
// ===== library: MasterCopy "APPLICATION_ID_READ_BLOCK" =====

FUNCTION_BLOCK "APPLICATION_ID_READ_BLOCK"   // FB5, SCL
{ S7_Optimized_Access := 'FALSE' }
VERSION : 0.1
   VAR_INPUT
      START_PARAMETER_READ : Bool;
      APPLICATION_ID : Int;
      PROFIdrive_OR_VACON_TELEGRAM_INPUT_ADDRESS : Int;
   END_VAR
   VAR_OUTPUT
      DONE : Bool;
      BUSY : Bool;
      ERROR : Bool;
      ERROR_CODE : DWord;
      VALUE : Int;
   END_VAR
   VAR
      PROFIdrive_param_read_request_record : Struct
         request_ref : Byte;
         request_id : Byte;
         axis_number : Byte;
         num_of_params_requested : Byte;
         attribute : Byte;
         num_of_elements : Byte;
         pnu : Int;
         subindex : Int;
      END_STRUCT;
      PROFIdrive_param_read_response : Struct
         request_ref : Byte;
         response_id : Byte;
         axis_number : Byte;
         num_of_parameters : Byte;
         format : Byte;
         num_of_values : Byte;
         value : Int;
      END_STRUCT;
      parameter_read_state : Int := 1;
      previous_start_parameter_read : Bool;
      stored_id : Int;
      stored_value : Int;
      WRREC_Instance : WRREC;
      stored_status : DWord;
      RDREC_Instance : RDREC;
      response_len : Int;
   END_VAR
   VAR_TEMP
      temp_done : Bool;
      temp_status : DWord;
      temp_error : Bool;
      temp_busy : Bool;
      temp_request_ref : Int;
      temp_valid : Bool;
      nooftries : Int;
   END_VAR
BEGIN
   CASE #parameter_read_state OF
       0:
           #parameter_read_state := 1;
           ;
       1:  // Statement section case 1
           IF #previous_start_parameter_read = 0 AND #START_PARAMETER_READ = 1 THEN
               #DONE := 0;
               #BUSY := 1;
               #ERROR := 0;
               #ERROR_CODE := 0;
               #nooftries := 0;
               #stored_id := #APPLICATION_ID;
               #PROFIdrive_param_read_request_record.attribute := 16#10;
               #PROFIdrive_param_read_request_record.axis_number := 1;
               #PROFIdrive_param_read_request_record.num_of_elements := 1;
               #PROFIdrive_param_read_request_record.num_of_params_requested := 1;
               #PROFIdrive_param_read_request_record.pnu := 10001;
               #PROFIdrive_param_read_request_record.request_id := 1; //change request, 1=read request
               #PROFIdrive_param_read_request_record.request_ref := INT_TO_CHAR(#temp_request_ref);
               #PROFIdrive_param_read_request_record.subindex := #stored_id;
               #temp_busy := 0;
               #temp_done := 0;
               #temp_error := 0;
               #temp_status := 0;
               #WRREC_Instance(REQ := 1,
                               ID := INT_TO_DWORD(#PROFIdrive_OR_VACON_TELEGRAM_INPUT_ADDRESS),
                               INDEX := 16#002f,
                               BUSY => #temp_busy,
                               DONE => #temp_done,
                               ERROR => #temp_error,
                               LEN := 10,
                               RECORD := #PROFIdrive_param_read_request_record,
                               STATUS => #stored_status);

               #parameter_read_state := 2; //start new parameter write sequence
           ELSE
               #parameter_read_state := 1;
               #DONE := 0;
               #BUSY := 0;
               #ERROR := 0;
               #ERROR_CODE := 0;
               #VALUE := 0;
           END_IF;
           ;
       2:  //check parameter write status
           #WRREC_Instance(REQ := 0,
                           ID := INT_TO_DWORD(#PROFIdrive_OR_VACON_TELEGRAM_INPUT_ADDRESS),
                           INDEX := 16#002f,
                           BUSY => #temp_busy,
                           DONE => #temp_done,
                           ERROR => #temp_error,
                           LEN := 10,
                           RECORD := #PROFIdrive_param_read_request_record,
                           STATUS => #stored_status);
           IF #temp_busy = 1 THEN
               // Statement section IF
               #parameter_read_state := 2; //check again next time
               #BUSY := 1;
               ;
           ELSIF #temp_done = 1 THEN
               #parameter_read_state := 3;
               #DONE := 0;
               #BUSY := 1;
               ;
           ELSIF #temp_error = 1 THEN
               #parameter_read_state := 20; //parameter write error state
               #ERROR := 1;
               #BUSY := 0;
               #ERROR_CODE := #stored_status;
           END_IF;
           ;

       3:  //Read response record
           #RDREC_Instance(REQ := 1,
                           ID := INT_TO_DWORD(#PROFIdrive_OR_VACON_TELEGRAM_INPUT_ADDRESS),
                           INDEX := 16#002f,
                           MLEN := 8,
                           BUSY => #temp_busy,
                           ERROR => #temp_error,
                           LEN => #response_len,
                           STATUS => #stored_status,
                           VALID => #temp_valid,
                           RECORD := #PROFIdrive_param_read_response);
           IF #temp_valid = 1 THEN
               // Statement section IF
               IF #PROFIdrive_param_read_response.format = 16#44 THEN
                   // Statement section IF
                   #parameter_read_state := 7; //done state
                   #DONE := 0;
                   #BUSY := 0;
                   #ERROR := 1;
                   #parameter_read_state := 30;
                   #VALUE := 0;
                   #ERROR_CODE := INT_TO_DWORD(#PROFIdrive_param_read_response.value);
                   #stored_status := #ERROR_CODE;
                   ;
               ELSE
                   #parameter_read_state := 7; //done state
                   #DONE := 1;
                   #BUSY := 0;
                   #VALUE := #PROFIdrive_param_read_response.value;
                   ;
               END_IF;
           ELSIF #temp_busy = 1 THEN
               #parameter_read_state := 3;
               #BUSY := 1;
               ;
           ELSIF #temp_error = 1 THEN
               IF #stored_status = 16#DE80B500 AND #nooftries < 10 THEN
                   #parameter_read_state := 4;
                   #DONE := 0;
                   #BUSY := 1;
                   #ERROR := 0;
                   #ERROR_CODE := 0;
                   #nooftries := #nooftries + 1;
                   ;
               ELSE
                   #parameter_read_state := 30;
                   #DONE := 0;
                   #BUSY := 0;
                   #ERROR := 1;
                   #ERROR_CODE := #stored_status;
                   ;
               END_IF;
               ;
           END_IF;
           ;
       4:
           //just a wait state when RDREC fails in state 3
           #parameter_read_state := 3;
           ;
       5:
           ;
       6:
           ;
       7:  // parameter write done state
           #DONE := 1;
           #BUSY := 0;
           #VALUE := #PROFIdrive_param_read_response.value;

           IF #START_PARAMETER_READ = 0 THEN
               // Statement section IF
               #parameter_read_state := 0;
               ;
           ELSE
               #parameter_read_state := 7;
           END_IF;

           ;
       20: //parameter write error state
           #BUSY := 0;
           #ERROR := 1;
           #DONE := 0;
           #ERROR_CODE := #stored_status;

           IF #START_PARAMETER_READ = 0 THEN
               // Statement section IF
               #parameter_read_state := 0;
               ;
           ELSE
               #parameter_read_state := 20;
           END_IF;

           ;
       30: //parameter write response error state
           #ERROR := 1;
           #ERROR_CODE := #stored_status;
           #DONE := 0;
           #BUSY := 0;

           IF #START_PARAMETER_READ = 0 THEN
               // Statement section IF
               #parameter_read_state := 0;
               ;
           ELSE
               #parameter_read_state := 30;
           END_IF;
           ;
       40:
           #BUSY := 0;
           #parameter_read_state := 40;
           ;
       ELSE  // Statement section ELSE
           ;
   END_CASE;
   #previous_start_parameter_read := #START_PARAMETER_READ;
END_FUNCTION_BLOCK

// ===== library: MasterCopy "APPLICATION_ID_WRITE_BLOCK" =====

FUNCTION_BLOCK "APPLICATION_ID_WRITE_BLOCK"   // FB4, SCL
{ S7_Optimized_Access := 'FALSE' }
VERSION : 0.1
   VAR_INPUT
      START_PARAMETER_WRITE : Bool;
      APPLICATION_ID : Int;
      VALUE : Int;
      PROFIdrive_OR_VACON_TELEGRAM_INPUT_ADDRESS : Int;
   END_VAR
   VAR_OUTPUT
      DONE : Bool;
      BUSY : Bool;
      ERROR : Bool;
      ERROR_CODE : DWord;
   END_VAR
   VAR
      WRREC_Instance : WRREC;
      RDREC_Instance : RDREC;
      parameter_write_state : Int := 1;
      PROFIdrive_param_write_request : Struct
         request_ref : Byte;
         request_id : Byte;
         axis_number : Byte;
         num_of_params_requested : Byte;
         attribute : Byte;
         num_of_elements : Byte;
         pnu : Int;
         subindex : Int;
         format : Byte;
         num_of_values : Byte;
         value : Int;
      END_STRUCT;
      previous_start_parameter_write : Bool;
      PROFIdrive_parameter_write_request_response : Struct
         request_ref : Byte;
         response_id : Byte;
         axis_number : Byte;
         num_of_params_affected : Byte;
         format : Byte;
         no_of_values : Byte;
         value : Int;
      END_STRUCT;
      stored_id : Int;
      stored_value : Int;
      response_len : Int;
      stored_status : DWord;
   END_VAR
   VAR_TEMP
      temp_busy : Bool;
      temp_done : Bool;
      temp_error : Bool;
      temp_status : DWord;
      temp_request_ref : Int;
      temp_valid : Bool;
      nooftries : Int;
   END_VAR
BEGIN
   CASE #parameter_write_state OF
       0:
           #parameter_write_state := 1;
           ;
       1:  // Statement section case 1
           IF #previous_start_parameter_write = 0 AND #START_PARAMETER_WRITE = 1 THEN
               #stored_id := #APPLICATION_ID;
               #stored_value := #VALUE;
               #DONE := 0;
               #BUSY := 1;
               #ERROR := 0;
               #ERROR_CODE := 0;
               #PROFIdrive_param_write_request.attribute := 16#10;
               #PROFIdrive_param_write_request.axis_number := 1;
               #PROFIdrive_param_write_request.format := 16#42; //word, 41=byte, 43=double word 
               #PROFIdrive_param_write_request.num_of_elements := 1;
               #PROFIdrive_param_write_request.num_of_params_requested := 1;
               #PROFIdrive_param_write_request.num_of_values := 1;
               #PROFIdrive_param_write_request.pnu := 10001;
               #PROFIdrive_param_write_request.request_id := 2; //change request, 1=read request
               #PROFIdrive_param_write_request.request_ref := INT_TO_CHAR(#temp_request_ref);
               #PROFIdrive_param_write_request.subindex := #stored_id;
               #PROFIdrive_param_write_request.value := #stored_value;
               #PROFIdrive_parameter_write_request_response.axis_number := 0;
               #PROFIdrive_parameter_write_request_response.format := 0;
               #PROFIdrive_parameter_write_request_response.no_of_values := 0;
               #PROFIdrive_parameter_write_request_response.num_of_params_affected := 0;
               #PROFIdrive_parameter_write_request_response.request_ref := 0;
               #PROFIdrive_parameter_write_request_response.response_id := 0;
               #PROFIdrive_parameter_write_request_response.value := 0;


               #temp_busy := 0;
               #temp_done := 0;
               #temp_error := 0;
               #temp_status := 0;
               #temp_valid := 0;
               #nooftries := 0;
               #WRREC_Instance(REQ := 1,
                               ID := INT_TO_DWORD(#PROFIdrive_OR_VACON_TELEGRAM_INPUT_ADDRESS),
                               INDEX := 16#002f,
                               BUSY => #temp_busy,
                               DONE => #temp_done,
                               ERROR => #temp_error,
                               LEN := 14,
                               RECORD := #PROFIdrive_param_write_request,
                               STATUS => #temp_status);
               #parameter_write_state := 2; //start new parameter write sequence
           ELSE
               #parameter_write_state := 1;
               #DONE := 0;
               #BUSY := 0;
               #ERROR := 0;
               #ERROR_CODE := 0;
           END_IF;
           ;
       2:  //check parameter write status
           #WRREC_Instance(REQ := 1,
                           ID := INT_TO_DWORD(#PROFIdrive_OR_VACON_TELEGRAM_INPUT_ADDRESS),
                           INDEX := 16#002f,
                           BUSY => #temp_busy,
                           DONE => #temp_done,
                           ERROR => #temp_error,
                           LEN := 14,
                           RECORD := #PROFIdrive_param_write_request,
                           STATUS => #stored_status);
           IF #temp_busy = 1 THEN
               // Statement section IF
               #parameter_write_state := 2; //check again next time
               #DONE := 0;
               #BUSY := 1;
               #ERROR := 0;
               #ERROR_CODE := 0;
               ;
           ELSIF #temp_done = 1 THEN
               #parameter_write_state := 3; //consider this a success
               #DONE := 0;
               #BUSY := 1;
               #ERROR := 0;
               #ERROR_CODE := 0;
               ;
           ELSIF #temp_error = 1 THEN
               #parameter_write_state := 20; //parameter write error state
               #ERROR := 1;
               #BUSY := 0;
               #DONE := 0;
               #ERROR_CODE := #stored_status;
           END_IF;

           ;
       3:  //parameter write ok state, read write response
           #RDREC_Instance(REQ:=1,
                           ID:=INT_TO_DWORD(#PROFIdrive_OR_VACON_TELEGRAM_INPUT_ADDRESS),
                           INDEX:=16#002f,
                           MLEN:=8,
                           BUSY => #temp_busy,
                           ERROR => #temp_error,
                           LEN => #response_len,
                           STATUS => #stored_status,
                           VALID => #temp_valid,
                           RECORD:=#PROFIdrive_parameter_write_request_response);
           IF #temp_valid = 1 THEN
       // Statement section IF
               IF #PROFIdrive_parameter_write_request_response.format = 68 THEN
                   // Statement section IF
                   #parameter_write_state := 20; //done state
                   #DONE := 0;
                   #BUSY := 0;
                   #ERROR := 1;
                   #stored_status := INT_TO_DWORD(#PROFIdrive_parameter_write_request_response.value);
                   #ERROR_CODE := 0;
                   ;
               ELSE
                   #parameter_write_state := 7; //done state
                   #DONE := 1;
                   #BUSY := 0;
                   #ERROR := 0;
                   #ERROR_CODE := 0;
                   ;
               END_IF;
           ;
           ELSIF #temp_busy = 1 THEN
               #parameter_write_state := 3;
               #DONE := 0;
               #BUSY := 1;
               #ERROR := 0;
               #ERROR_CODE := 0;
           ;
           ELSIF #temp_error = 1 THEN
               IF #stored_status = 16#DE80B500 AND #nooftries < 10 THEN
                   #parameter_write_state := 4;
                   #DONE := 0;
                   #BUSY := 1;
                   #ERROR := 0;
                   #ERROR_CODE := 0;
                   #nooftries := #nooftries + 1;
                   ;
               ELSE
                   #parameter_write_state := 30;
                   #DONE := 0;
                   #BUSY := 0;
                   #ERROR := 1;
                   #ERROR_CODE := #stored_status;
                   ;
               END_IF;
               ;
           END_IF;

           ;
       4:
           //just a wait state when RDREC fails in state 3
           #parameter_write_state := 3;
           ;
       5:
           ;
       6:
           ;
       7:  // parameter write done state
           #DONE := 1;
           #BUSY := 0;
           #ERROR := 0;
           #ERROR_CODE := 0;
           IF #START_PARAMETER_WRITE = 0 THEN
               // Statement section IF
               #parameter_write_state := 1;
               ;
           ELSE
               #parameter_write_state := 7;
           END_IF;
           ;
       20: //parameter write error state
           #DONE := 0;
           #BUSY := 0;
           #ERROR := 1;
           #ERROR_CODE := #stored_status;

           IF #START_PARAMETER_WRITE = 0 THEN
               // Statement section IF
               #parameter_write_state := 1;
               ;
           ELSE
               #parameter_write_state := 20;
           END_IF;
           ;
       30: //parameter write response error state
           #DONE := 0;
           #BUSY := 0;
           #ERROR := 1;
           #ERROR_CODE := #stored_status;

           IF #START_PARAMETER_WRITE = 0 THEN
               // Statement section IF
               #parameter_write_state := 1;
               ;
           ELSE
               #parameter_write_state := 30;
           END_IF;
           ;
       40:
           #BUSY := 0;
           #parameter_write_state := 40;
           ;
       ELSE  // Statement section ELSE
           ;
   END_CASE;
   #previous_start_parameter_write := #START_PARAMETER_WRITE;
END_FUNCTION_BLOCK

// ===== library: MasterCopy "PROFIdrive_CONTROL_BLOCK_OPTE3_OPTE5" =====

FUNCTION_BLOCK "PROFIdrive_CONTROL_BLOCK_OPTE3_OPTE5"   // FB2, SCL
{ S7_Optimized_Access := 'FALSE' }
VERSION : 0.1
   VAR_INPUT
      RUN : Bool;
      DIRECTION : Bool;
      QUICK_STOP : Bool;
      FAULT_RESET : Bool;
      SPEED_REFERENCE : Int;
      PROFIdrive_ST1_INPUT_ADDRESS : Int;
      PROFIDrive_ST1_OUTPUT_ADDRESS : Int;
   END_VAR
   VAR_OUTPUT
      RUNNING : Bool;
      FAULT_PRESENT : Bool;
      SPEED_ACTUAL : Int;
      CURRENT_DIRECTION : Bool;
      READY : Bool;
      AT_REFERENCE : Bool;
   END_VAR
   VAR_TEMP
      PROFIdrive_ZSW2 : Word;
      PROFIdrive_ZSW2_BIT AT PROFIdrive_ZSW2 : Array[0..15] of Bool;
      PROFIdrive_STW2 : Word;
      PROFIdrive_STW2_BIT AT PROFIdrive_STW2 : Array[0..15] of Bool;
      PROFIdrive_speed_reference : Int;
      PROFIdrive_actual_speed : Int;
      SPEED_CALC_TEMP : DInt;
   END_VAR
BEGIN
   #PROFIdrive_STW2 := 16#0476; (**)
   #PROFIdrive_ZSW2 := %IW(#PROFIdrive_ST1_INPUT_ADDRESS):P;
   #PROFIdrive_actual_speed := %IW(#PROFIdrive_ST1_INPUT_ADDRESS + 2):P;

   IF #RUN = TRUE AND #QUICK_STOP = FALSE THEN
       // Statement section IF
       IF #PROFIdrive_ZSW2_BIT[14] = TRUE THEN
           #PROFIdrive_STW2_BIT[8] := FALSE;
       ELSIF  #PROFIdrive_ZSW2_BIT[8] = TRUE AND #PROFIdrive_ZSW2_BIT[9] = FALSE AND #PROFIdrive_ZSW2_BIT[11] = FALSE AND #PROFIdrive_ZSW2_BIT[14] = FALSE THEN
           // Statement section IF
           #PROFIdrive_STW2_BIT[8] := TRUE;
       ELSIF  #PROFIdrive_ZSW2_BIT[8] = TRUE AND #PROFIdrive_ZSW2_BIT[9] = TRUE AND #PROFIdrive_ZSW2_BIT[10] = FALSE AND #PROFIdrive_ZSW2_BIT[14] = FALSE THEN
           #PROFIdrive_STW2_BIT[8] := TRUE;
           #PROFIdrive_STW2_BIT[11] := TRUE;
       ELSE
           #PROFIdrive_STW2_BIT[11] := TRUE;
           #PROFIdrive_STW2_BIT[8] := TRUE;
       END_IF;
   ELSIF #RUN = FALSE AND #QUICK_STOP = FALSE THEN
       #PROFIdrive_STW2_BIT[11] := FALSE;
       #PROFIdrive_STW2_BIT[8] := TRUE;
   ELSIF #QUICK_STOP = TRUE AND #RUN = TRUE THEN
       #PROFIdrive_STW2_BIT[10] := FALSE;
       #PROFIdrive_STW2_BIT[8] := TRUE;
       #PROFIdrive_STW2_BIT[11] := TRUE;
   END_IF;

   IF #FAULT_RESET = TRUE THEN
       #PROFIdrive_STW2_BIT[15] := TRUE;
   ELSE
       #PROFIdrive_STW2_BIT[15] := FALSE;
   END_IF;

   IF #PROFIdrive_ZSW2_BIT[11] = TRUE THEN
       // Statement section IF
       #FAULT_PRESENT := TRUE;
   ELSE
       #FAULT_PRESENT := FALSE;
   END_IF;

   IF #PROFIdrive_ZSW2_BIT[4] = TRUE THEN
       // Statement section IF
       #RUNNING := TRUE;
   ELSE
       #RUNNING := FALSE;
   END_IF;

   IF #PROFIdrive_ZSW2_BIT[5] = TRUE THEN
       // Statement section IF
       #READY := TRUE;
   ELSE
       #READY := FALSE;
       ;
   END_IF;

   IF #PROFIdrive_ZSW2_BIT[0] = TRUE THEN
       // Statement section IF
       #AT_REFERENCE := TRUE;
       ;
   ELSE
       #AT_REFERENCE := FALSE;
       ;
   END_IF;


   IF #DIRECTION = FALSE THEN
       #SPEED_CALC_TEMP := #SPEED_REFERENCE;
       #SPEED_CALC_TEMP := (16384 * #SPEED_CALC_TEMP) / 10000;
       #PROFIdrive_speed_reference := DINT_TO_INT(#SPEED_CALC_TEMP);
   ELSE
       #SPEED_CALC_TEMP := #SPEED_REFERENCE;
       #SPEED_CALC_TEMP := (-(16384 * #SPEED_CALC_TEMP)) / 10000;
       #PROFIdrive_speed_reference := DINT_TO_INT(#SPEED_CALC_TEMP);
   END_IF;

   IF #PROFIdrive_actual_speed < 0 THEN
       // Statement section IF
       #SPEED_CALC_TEMP := #PROFIdrive_actual_speed;
       #SPEED_CALC_TEMP := (-(#SPEED_CALC_TEMP) * 10000) / 16384;
       #SPEED_ACTUAL := DINT_TO_INT(#SPEED_CALC_TEMP);
       #CURRENT_DIRECTION := TRUE;
   ELSE
       #SPEED_CALC_TEMP := #PROFIdrive_actual_speed;
       #SPEED_CALC_TEMP := (#SPEED_CALC_TEMP * 10000) / 16384;
       #SPEED_ACTUAL := DINT_TO_INT(#SPEED_CALC_TEMP);
       #CURRENT_DIRECTION := FALSE;
   END_IF;

   %QW(#PROFIDrive_ST1_OUTPUT_ADDRESS):P := #PROFIdrive_STW2;
   %QW(#PROFIDrive_ST1_OUTPUT_ADDRESS + 2):P := #PROFIdrive_speed_reference;
END_FUNCTION_BLOCK

// ===== library: MasterCopy "PROFIdrive_CONTROL_BLOCK_OPTE3_OPTE5_8PD" =====

FUNCTION_BLOCK "PROFIdrive_CONTROL_BLOCK_OPTE3_OPTE5_8PD"   // FB7, SCL
{ S7_Optimized_Access := 'FALSE' }
VERSION : 0.1
   VAR_INPUT
      RUN : Bool;
      DIRECTION : Bool;
      QUICK_STOP : Bool;
      FAULT_RESET : Bool;
      SPEED_REFERENCE : Int;
      PROFIdrive_ST1_INPUT_ADDRESS : Int;
      PROFIDrive_ST1_OUTPUT_ADDRESS : Int;
   END_VAR
   VAR_OUTPUT
      RUNNING : Bool;
      FAULT_PRESENT : Bool;
      SPEED_ACTUAL : Int;
      CURRENT_DIRECTION : Bool;
      READY : Bool;
      AT_REFERENCE : Bool;
      PD1_OUT : Int;
      PD2_OUT : Int;
      PD3_OUT : Int;
      PD4_OUT : Int;
      PD5_OUT : Int;
      PD6_OUT : Int;
      PD7_OUT : Int;
      PD8_OUT : Int;
   END_VAR
   VAR_TEMP
      PROFIdrive_ZSW2 : Word;
      PROFIdrive_ZSW2_BIT AT PROFIdrive_ZSW2 : Array[0..15] of Bool;
      PROFIdrive_STW2 : Word;
      PROFIdrive_STW2_BIT AT PROFIdrive_STW2 : Array[0..15] of Bool;
      PROFIdrive_speed_reference : Int;
      PROFIdrive_actual_speed : Int;
      SPEED_CALC_TEMP : DInt;
   END_VAR
BEGIN
   #PROFIdrive_STW2 := 16#0476; (**)
   #PROFIdrive_ZSW2 := %IW(#PROFIdrive_ST1_INPUT_ADDRESS):P;
   #PROFIdrive_actual_speed := %IW(#PROFIdrive_ST1_INPUT_ADDRESS + 2):P;
   #PD1_OUT := WORD_TO_INT(%IW(#PROFIdrive_ST1_INPUT_ADDRESS + 4):P);
   #PD2_OUT := WORD_TO_INT(%IW(#PROFIdrive_ST1_INPUT_ADDRESS + 6):P);
   #PD3_OUT := WORD_TO_INT(%IW(#PROFIdrive_ST1_INPUT_ADDRESS + 8):P);
   #PD4_OUT := WORD_TO_INT(%IW(#PROFIdrive_ST1_INPUT_ADDRESS + 10):P);
   #PD5_OUT := WORD_TO_INT(%IW(#PROFIdrive_ST1_INPUT_ADDRESS + 12):P);
   #PD6_OUT := WORD_TO_INT(%IW(#PROFIdrive_ST1_INPUT_ADDRESS + 14):P);
   #PD7_OUT := WORD_TO_INT(%IW(#PROFIdrive_ST1_INPUT_ADDRESS + 16):P);
   #PD8_OUT := WORD_TO_INT(%IW(#PROFIdrive_ST1_INPUT_ADDRESS + 18):P);

   IF #RUN = TRUE AND #QUICK_STOP = FALSE THEN
       // Statement section IF
       IF #PROFIdrive_ZSW2_BIT[14] = TRUE THEN
           #PROFIdrive_STW2_BIT[8] := FALSE;
       ELSIF  #PROFIdrive_ZSW2_BIT[8] = TRUE AND #PROFIdrive_ZSW2_BIT[9] = FALSE AND #PROFIdrive_ZSW2_BIT[11] = FALSE AND #PROFIdrive_ZSW2_BIT[14] = FALSE THEN
           // Statement section IF
           #PROFIdrive_STW2_BIT[8] := TRUE;
       ELSIF  #PROFIdrive_ZSW2_BIT[8] = TRUE AND #PROFIdrive_ZSW2_BIT[9] = TRUE AND #PROFIdrive_ZSW2_BIT[10] = FALSE AND #PROFIdrive_ZSW2_BIT[14] = FALSE THEN
           #PROFIdrive_STW2_BIT[8] := TRUE;
           #PROFIdrive_STW2_BIT[11] := TRUE;
       ELSE
           #PROFIdrive_STW2_BIT[11] := TRUE;
           #PROFIdrive_STW2_BIT[8] := TRUE;
       END_IF;
   ELSIF #RUN = FALSE AND #QUICK_STOP = FALSE THEN
       #PROFIdrive_STW2_BIT[11] := FALSE;
       #PROFIdrive_STW2_BIT[8] := TRUE;
   ELSIF #QUICK_STOP = TRUE AND #RUN = TRUE THEN
       #PROFIdrive_STW2_BIT[10] := FALSE;
       #PROFIdrive_STW2_BIT[8] := TRUE;
       #PROFIdrive_STW2_BIT[11] := TRUE;
   END_IF;

   IF #FAULT_RESET = TRUE THEN
       #PROFIdrive_STW2_BIT[15] := TRUE;
   ELSE
       #PROFIdrive_STW2_BIT[15] := FALSE;
   END_IF;

   IF #PROFIdrive_ZSW2_BIT[11] = TRUE THEN
       // Statement section IF
       #FAULT_PRESENT := TRUE;
   ELSE
       #FAULT_PRESENT := FALSE;
   END_IF;

   IF #PROFIdrive_ZSW2_BIT[4] = TRUE THEN
       // Statement section IF
       #RUNNING := TRUE;
   ELSE
       #RUNNING := FALSE;
   END_IF;

   IF #PROFIdrive_ZSW2_BIT[5] = TRUE THEN
       // Statement section IF
       #READY := TRUE;
   ELSE
       #READY := FALSE;
       ;
   END_IF;

   IF #PROFIdrive_ZSW2_BIT[0] = TRUE THEN
       // Statement section IF
       #AT_REFERENCE := TRUE;
       ;
   ELSE
       #AT_REFERENCE := FALSE;
       ;
   END_IF;


   IF #DIRECTION = FALSE THEN
       #SPEED_CALC_TEMP := #SPEED_REFERENCE;
       #SPEED_CALC_TEMP := (16384 * #SPEED_CALC_TEMP) / 10000;
       #PROFIdrive_speed_reference := DINT_TO_INT(#SPEED_CALC_TEMP);
   ELSE
       #SPEED_CALC_TEMP := #SPEED_REFERENCE;
       #SPEED_CALC_TEMP := (-(16384 * #SPEED_CALC_TEMP)) / 10000;
       #PROFIdrive_speed_reference := DINT_TO_INT(#SPEED_CALC_TEMP);
   END_IF;

   IF #PROFIdrive_actual_speed < 0 THEN
       // Statement section IF
       #SPEED_CALC_TEMP := #PROFIdrive_actual_speed;
       #SPEED_CALC_TEMP := (-(#SPEED_CALC_TEMP) * 10000) / 16384;
       #SPEED_ACTUAL := DINT_TO_INT(#SPEED_CALC_TEMP);
       #CURRENT_DIRECTION := TRUE;
   ELSE
       #SPEED_CALC_TEMP := #PROFIdrive_actual_speed;
       #SPEED_CALC_TEMP := (#SPEED_CALC_TEMP * 10000) / 16384;
       #SPEED_ACTUAL := DINT_TO_INT(#SPEED_CALC_TEMP);
       #CURRENT_DIRECTION := FALSE;
   END_IF;

   %QW(#PROFIDrive_ST1_OUTPUT_ADDRESS):P := #PROFIdrive_STW2;
   %QW(#PROFIDrive_ST1_OUTPUT_ADDRESS + 2):P := #PROFIdrive_speed_reference;
END_FUNCTION_BLOCK

// ===== library: MasterCopy "VACON_CONTROL_BLOCK" =====

FUNCTION_BLOCK "VACON_CONTROL_BLOCK"   // FB6, SCL
{ S7_Optimized_Access := 'FALSE' }
VERSION : 0.1
   VAR_INPUT
      RUN : Bool;
      DIRECTION : Bool;
      FAULT_RESET : Bool;
      SPEED_REFERENCE : Int;
      VENDOR_TELEGRAM1_INPUT_ADDRESS : Int;
      VENDOR_TELEGRAM1_OUTPUT_ADDRESS : Int;
   END_VAR
   VAR_OUTPUT
      RUNNING : Bool;
      FAULT_PRESENT : Bool;
      SPEED_ACTUAL : Int;
      CURRENT_DIRECTION : Bool;
      READY : Bool;
      AT_REFERENCE : Bool;
   END_VAR
   VAR_TEMP
      Vacon_FBFixedControlWord : Word;
      Vacon_FBFixedControlWord_BIT AT Vacon_FBFixedControlWord : Array[0..15] of Bool;
      Vacon_FBFixedStatusWord : Word;
      Vacon_FBFixedStatusWord_BITS AT Vacon_FBFixedStatusWord : Array[0..15] of Bool;
      Vacon_Speed_Actual : Int;
   END_VAR
BEGIN
   #Vacon_FBFixedStatusWord := %IW(#VENDOR_TELEGRAM1_INPUT_ADDRESS):P;
   #Vacon_FBFixedControlWord := 16#03;
   #Vacon_Speed_Actual := %IW(#VENDOR_TELEGRAM1_INPUT_ADDRESS + 2):P;
   IF #RUN = 1 THEN
       // Statement section IF
       #Vacon_FBFixedControlWord_BIT[8] := 1;
   ELSE
       #Vacon_FBFixedControlWord_BIT[8] := 0;
       ;
   END_IF;

   IF #DIRECTION = 1 THEN
       #Vacon_FBFixedControlWord_BIT[9] := 1;
       ;
   ELSE
       #Vacon_FBFixedControlWord_BIT[9] := 0;
       ;
   END_IF;

   IF #FAULT_RESET = 1 THEN
       // Statement section IF
       #Vacon_FBFixedControlWord_BIT[10] := 1;
       ;
   ELSE
       #Vacon_FBFixedControlWord_BIT[10] := 0;
   END_IF;

   IF #Vacon_FBFixedStatusWord_BITS[10] = 1 THEN
       // Statement section IF
       #CURRENT_DIRECTION := 1;
   ELSE
       #CURRENT_DIRECTION := 0;
       ;
   END_IF;

   IF #Vacon_FBFixedStatusWord_BITS[9] = 1 THEN
       // Statement section IF
       #RUNNING := 1;
   ELSE
       #RUNNING := 0;
       ;
   END_IF;

   IF #Vacon_FBFixedStatusWord_BITS[11] = 1 THEN
       // Statement section IF
       #FAULT_PRESENT := 1;
   ELSE
       #FAULT_PRESENT := 0;
       ;
   END_IF;

   IF #Vacon_FBFixedStatusWord_BITS[8] = TRUE THEN
       // Statement section IF
       #READY := TRUE;
   ELSE
       #READY := FALSE
       ;
   END_IF;

   IF #Vacon_FBFixedStatusWord_BITS[13] THEN
       // Statement section IF
       #AT_REFERENCE := 1;
   ELSE
       #AT_REFERENCE := 0;
       ;
   END_IF;



   %QW(#VENDOR_TELEGRAM1_OUTPUT_ADDRESS):P := #Vacon_FBFixedControlWord;
   %QW(#VENDOR_TELEGRAM1_OUTPUT_ADDRESS+2):P := #SPEED_REFERENCE;
   #SPEED_ACTUAL := #Vacon_Speed_Actual;
END_FUNCTION_BLOCK

// ===== library: MasterCopy "VACON_CONTROL_BLOCK_8PD" =====

FUNCTION_BLOCK "VACON_CONTROL_BLOCK_8PD"   // FB3, SCL
{ S7_Optimized_Access := 'FALSE' }
VERSION : 0.1
   VAR_INPUT
      RUN : Bool;
      DIRECTION : Bool;
      FAULT_RESET : Bool;
      SPEED_REFERENCE : Int;
      VENDOR_TELEGRAM1_INPUT_ADDRESS : Int;
      VENDOR_TELEGRAM1_OUTPUT_ADDRESS : Int;
   END_VAR
   VAR_OUTPUT
      RUNNING : Bool;
      FAULT_PRESENT : Bool;
      SPEED_ACTUAL : Int;
      CURRENT_DIRECTION : Bool;
      READY : Bool;
      AT_REFERENCE : Bool;
      PD1_OUT : Int;
      PD2_OUT : Int;
      PD3_OUT : Int;
      PD4_OUT : Int;
      PD5_OUT : Int;
      PD6_OUT : Int;
      PD7_OUT : Int;
      PD8_OUT : Int;
   END_VAR
   VAR_TEMP
      Vacon_FBFixedControlWord : Word;
      Vacon_FBFixedControlWord_BIT AT Vacon_FBFixedControlWord : Array[0..15] of Bool;
      Vacon_FBFixedStatusWord : Word;
      Vacon_FBFixedStatusWord_BITS AT Vacon_FBFixedStatusWord : Array[0..15] of Bool;
      Vacon_Speed_Actual : Int;
   END_VAR
BEGIN
   #Vacon_FBFixedStatusWord := %IW(#VENDOR_TELEGRAM1_INPUT_ADDRESS):P;
   #Vacon_FBFixedControlWord := 16#03;
   #Vacon_Speed_Actual := %IW(#VENDOR_TELEGRAM1_INPUT_ADDRESS + 2):P;
   #PD1_OUT := WORD_TO_INT(%IW(#VENDOR_TELEGRAM1_INPUT_ADDRESS + 4):P);
   #PD2_OUT := WORD_TO_INT(%IW(#VENDOR_TELEGRAM1_INPUT_ADDRESS + 6):P);
   #PD3_OUT := WORD_TO_INT(%IW(#VENDOR_TELEGRAM1_INPUT_ADDRESS + 8):P);
   #PD4_OUT := WORD_TO_INT(%IW(#VENDOR_TELEGRAM1_INPUT_ADDRESS + 10):P);
   #PD5_OUT := WORD_TO_INT(%IW(#VENDOR_TELEGRAM1_INPUT_ADDRESS + 12):P);
   #PD6_OUT := WORD_TO_INT(%IW(#VENDOR_TELEGRAM1_INPUT_ADDRESS + 14):P);
   #PD7_OUT := WORD_TO_INT(%IW(#VENDOR_TELEGRAM1_INPUT_ADDRESS + 16):P);
   #PD8_OUT := WORD_TO_INT(%IW(#VENDOR_TELEGRAM1_INPUT_ADDRESS + 18):P);

   IF #RUN = 1 THEN
       // Statement section IF
       #Vacon_FBFixedControlWord_BIT[8] := 1;
   ELSE
       #Vacon_FBFixedControlWord_BIT[8] := 0;
       ;
   END_IF;

   IF #DIRECTION = 1 THEN
       #Vacon_FBFixedControlWord_BIT[9] := 1;
       ;
   ELSE
       #Vacon_FBFixedControlWord_BIT[9] := 0;
       ;
   END_IF;

   IF #FAULT_RESET = 1 THEN
       // Statement section IF
       #Vacon_FBFixedControlWord_BIT[10] := 1;
       ;
   ELSE
       #Vacon_FBFixedControlWord_BIT[10] := 0;
   END_IF;

   IF #Vacon_FBFixedStatusWord_BITS[10] = 1 THEN
       // Statement section IF
       #CURRENT_DIRECTION := 1;
   ELSE
       #CURRENT_DIRECTION := 0;
       ;
   END_IF;

   IF #Vacon_FBFixedStatusWord_BITS[9] = 1 THEN
       // Statement section IF
       #RUNNING := 1;
   ELSE
       #RUNNING := 0;
       ;
   END_IF;

   IF #Vacon_FBFixedStatusWord_BITS[11] = 1 THEN
       // Statement section IF
       #FAULT_PRESENT := 1;
   ELSE
       #FAULT_PRESENT := 0;
       ;
   END_IF;

   IF #Vacon_FBFixedStatusWord_BITS[8] = TRUE THEN
       // Statement section IF
       #READY := TRUE;
   ELSE
       #READY := FALSE
       ;
   END_IF;

   IF #Vacon_FBFixedStatusWord_BITS[13] THEN
       // Statement section IF
       #AT_REFERENCE := 1;
   ELSE
       #AT_REFERENCE := 0;
       ;
   END_IF;



   %QW(#VENDOR_TELEGRAM1_OUTPUT_ADDRESS):P := #Vacon_FBFixedControlWord;
   %QW(#VENDOR_TELEGRAM1_OUTPUT_ADDRESS+2):P := #SPEED_REFERENCE;
   #SPEED_ACTUAL := #Vacon_Speed_Actual;
END_FUNCTION_BLOCK